TYPE MultiAxis_Output_typ :
	STRUCT
		monitor 	: MultiAxis_monitor_typ ;
		Status		: MultiAxis_Statuses_typ ;
		Error		: MultiAxis_Error_typ ;
		
	END_STRUCT
END_TYPE

(* stored: Version 1.1.0.1, ProductVersion 3.1.4024.3
   DUT MultiAxis_Output_typ: Id {3658f95a-2344-0449-1ac2-69d97c08f4d0} *)
